TYPE ControlBESSparams :
STRUCT
END_STRUCT
END_TYPE

(* stored: Version 1.1.0.1, ProductVersion 3.1.4024.4
   DUT ControlBESSparams: Id {f466bd77-6e61-4b53-b1ea-2316ca608666} *)
